// TIA Portal V17 export
// export: Created 2022-04-06T07:28:40.5303201Z, ExportSetting WithDefaults, DisplayName Totally Integrated Automation Portal, DisplayVersion V17, DisplayName TIA Portal Openness, DisplayVersion V17, DisplayName TIA Portal Version Control Interface, DisplayVersion V17, DisplayName TIA Portal Test Suite Advanced, DisplayVersion V17, DisplayName SINAMICS Startdrive Advanced, DisplayVersion V17, DisplayName SINAMICS Startdrive G130, G150, S120, S150, SINAMICS MV, S210, DisplayVersion V17, DisplayName SINAMICS Startdrive G110M, G120, G120C, G120D, G120P, G115D, DisplayVersion V17, DisplayName STEP 7 Professional, DisplayVersion V17, DisplayName STEP 7 Safety, DisplayVersion V17, DisplayName WinCC Advanced / Unified PC, DisplayVersion V17
TYPE "LDrvSafe_typeSinaTlg901Control"
TITLE = LDrvSafe_typeSinaTlg901Control
// Failsafe user-defined data type for PROFIsafe telegram 901 to control the Safety Integrated Functions of SINAMICS
// stored: IsFailsafeCompliant true
   STRUCT
      STO { ExternalWritable := 'False'} : Bool;   // Safety Function Safe Torque Off
      SS1 { ExternalWritable := 'False'} : Bool;   // Safety Function Safe Stop 1
      SS2 { ExternalWritable := 'False'} : Bool;   // Safety Function Safe Stop 2
      SOS { ExternalWritable := 'False'} : Bool;   // Safety Function Safe Operating Stop
      SLS { ExternalWritable := 'False'} : Bool;   // Safety Function Safely-limited Speed
      reserved1 { ExternalWritable := 'False'} : Bool;   // Reserve bit 1
      SLP { ExternalWritable := 'False'} : Bool;   // Safety Function Safely-limited Position
      internalEventAcknowledge { ExternalWritable := 'False'} : Bool;   // Acknowledge Safety errors in the drive
      SLA { ExternalWritable := 'False'} : Bool;   // Safety Function Safely-limited Acceleration
      selectSLSbit0 { ExternalWritable := 'False'} : Bool;   // Select one of the the four SLS limits; operates together with bit 1
      selectSLSbit1 { ExternalWritable := 'False'} : Bool;   // Select one of the the four SLS limits; operates together with bit 0
      reserved2 { ExternalWritable := 'False'} : Bool;   // Reserve bit 2
      SDIpositive { ExternalWritable := 'False'} : Bool;   // Safety Function Safe Direction (positive direction)
      SDInegative { ExternalWritable := 'False'} : Bool;   // Safety Function Safe Direction (negative direction)
      reserved4 { ExternalWritable := 'False'} : Bool;   // Reserve bit 4
      reserved5 { ExternalWritable := 'False'} : Bool;   // Reserve bit 5
      reserved6 { ExternalWritable := 'False'} : Bool;   // Reserve bit 6
      reserved7 { ExternalWritable := 'False'} : Bool;   // Reserve bit 7
      reserved8 { ExternalWritable := 'False'} : Bool;   // Reserve bit 8
      selectSLPrange { ExternalWritable := 'False'} : Bool;   // Select one of the two SLP ranges
      reserved9 { ExternalWritable := 'False'} : Bool;   // Reserve bit 9
      reserved10 { ExternalWritable := 'False'} : Bool;   // Reserve bit 10
      reserved11 { ExternalWritable := 'False'} : Bool;   // Reserve bit 11
      SCA { ExternalWritable := 'False'} : Bool;   // Safety Function Safe Cam
      selectGearboxStageBit0 { ExternalWritable := 'False'} : Bool;   // Select one of the the eight gearbox stages; operates together with bit 1 and 2
      selectGearboxStageBit1 { ExternalWritable := 'False'} : Bool;   // Select one of the the eight gearbox stages; operates together with bit 0 and 2
      selectGearboxStageBit2 { ExternalWritable := 'False'} : Bool;   // Select one of the the eight gearbox stages; operates together with bit 0 and 1
      switchoverGearboxStage { ExternalWritable := 'False'} : Bool;   // Higher position tolerance at gearbox switching
      SS2E { ExternalWritable := 'False'} : Bool;   // Safety Function Safe Stop 2 with external stop
      reserved13 { ExternalWritable := 'False'} : Bool;   // Reserve bit 13
      reserved14 { ExternalWritable := 'False'} : Bool;   // Reserve bit 14
      reserved15 { ExternalWritable := 'False'} : Bool;   // Reserve bit 15
      variableSLS { ExternalWritable := 'False'} : Int;   // SLS limit 1 can be varied within 1 and 32.767 (0.03 and 100%)
   END_STRUCT;
END_TYPE
